FUNCTION_BLOCK MultiAgentSystemConnector (* JADE WORKER *)
  (* Standard: 61499-1 *)
  (* Version 1.0, 2014-04-22, Ahmed, Fraunhofer IGD *)
  (* Compiler header: package fb.rt; *)
  (* Compiler Java Sun JDK 1.5.0 *)
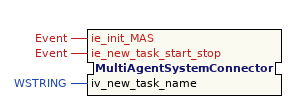
  EVENT_INPUT
    ie_init_MAS;
    ie_new_task_start_stop;
  END_EVENT
  VAR_INPUT
    iv_new_task_name : WSTRING;
  END_VAR
END_FUNCTION_BLOCK
